   VAR
      sUDT_HMIStatus { ExternalAccessible := 'False'; ExternalVisible := 'False'; ExternalWritable := 'False'; S7_SetPoint := 'False'} : "UDT_WE01Status";   // UDT Weigghing Scale status
      sUDT_Status { ExternalAccessible := 'False'; ExternalVisible := 'False'; ExternalWritable := 'False'; S7_SetPoint := 'False'} : "UDT_CommonStatus";   //  Common status structure
      sUDT_CommonStatus { ExternalAccessible := 'False'; ExternalVisible := 'False'; ExternalWritable := 'False'; S7_SetPoint := 'False'} : "UDT_CommonStatus";   //  Common status structure
      sUDT_CommonStatusOld { ExternalAccessible := 'False'; ExternalVisible := 'False'; ExternalWritable := 'False'; S7_SetPoint := 'False'} : "UDT_CommonStatus";   //  Auxiliary status structure
      sFB_TimerOnOffDelayAutoOn { ExternalAccessible := 'False'; ExternalVisible := 'False'; ExternalWritable := 'False'; S7_SetPoint := 'False'} : "FB_TimerOnOffDelay";
      sx_AutoOnDelayed { ExternalAccessible := 'False'; ExternalVisible := 'False'; ExternalWritable := 'False'} : Bool;
   END_VAR

   VAR CONSTANT
      cdi_DelayOffAutomaticOn : UDInt := 600000;   // Delay before turning off the AutoOn signal
   END_VAR


BEGIN
	(*
	----------------------------------------------------------------------------------------

	Version history:
	Date        | Version   | Author        | Remark
	----------------------------------------------------------------------------------------
	17/09/2019  | 2.0       | M.Singh       | first release TIA 15.1
	21/02/2023  | 4.0       | F.Baten       | 4.0 Release TIA 17.5
	12/03/2024  | 4.1       | S. Nieswie    | Variable name changes accroding to current standard

	 *)

	REGION 1 - Reset Error
	    // If reset Provided from outside; reset the Error

	    IF #iqUDT_EquipmentControl.Command.Reset THEN
	        #sUDT_HMIStatus.Specific.WeighingScaleFault := FALSE;
	    END_IF;
	END_REGION

	REGION 2 - Fault monitoring
	    // Make Camera Error Status

	    IF #ix_ScaleInFault THEN
	        #sUDT_HMIStatus.Specific.WeighingScaleFault := True;
	    END_IF;
	END_REGION

	REGION 3 - Send Automatic Signal to Weighing Scale
	    //  Delay the Turning off of "Automatic on" Signal to Weighing Scale
	    #sFB_TimerOnOffDelayAutoOn(iudi_OffDelayTime := #cdi_DelayOffAutomaticOn,
	                               ix_SignalToDelay := #iqUDT_EquipmentControl.Command.AutomaticOn,
	                               qx_DelayedSignal => #sx_AutoOnDelayed);

	    #qx_Automatic := #sx_AutoOnDelayed;
	END_REGION

	REGION 10 - Make Status
	    // Set Common Status Report

	    // Error active
	    #sUDT_CommonStatus.Error := #sUDT_HMIStatus.Specific.WeighingScaleFault;

	    // Running
	    #sUDT_CommonStatus.Running := #iqUDT_EquipmentControl.Command.AutomaticOn AND NOT #sUDT_CommonStatus.Error;

	    // Stopped
	    #sUDT_CommonStatus.Stopped := NOT #qx_Automatic;

	    IF #sUDT_CommonStatusOld <> #sUDT_CommonStatus                   // update on change
	    THEN

	        // HMI status initialization
	        #sUDT_HMIStatus.Status := 0;

	        // Running in Automatic mode
	        IF #sUDT_CommonStatus.Running
	        THEN
	            #sUDT_HMIStatus.Status := "DB_HMIStatusConfiguration".Running;
	        END_IF;

	        // Stopped
	        IF #sUDT_CommonStatus.Stopped THEN
	            #sUDT_HMIStatus.Status := "DB_HMIStatusConfiguration".Stopped;
	        END_IF;

	        // Error
	        IF #sUDT_HMIStatus.Specific.WeighingScaleFault
	        THEN
	            #sUDT_HMIStatus.Status := "DB_HMIStatusConfiguration".Error;
	        END_IF;

	        #sUDT_CommonStatusOld := #sUDT_CommonStatus;                  // Copy status to memory
	        #sUDT_Status := #sUDT_CommonStatus;                           // Copy status to output
	    END_IF;

	    #qUDT_HMIStatus := #sUDT_HMIStatus;                               // Copy HMI status to output
	    #qUDT_Status := #sUDT_Status;                                     // Copy common status to output


	END_REGION

	REGION 11 - Report to control block

	    // Function to manage report between control block and conveyor block

	    "FC_EquipmentReport"(iUDT_Status := #sUDT_CommonStatus,
	                         iqUDT_Control := #iqUDT_EquipmentControl);

	END_REGION


END_FUNCTION_BLOCK

FUNCTION_BLOCK "FB_MCOConveyLinxAixFullZPA"
TITLE = ConveyLinx reduced ZPA segment
{ S7_Optimized_Access := 'TRUE' }
AUTHOR : 'Ihab Ajram'
FAMILY : ConveyLinx
NAME : ConveyLinx_Reduced_ZPA
VERSION : 0.6
//Version
//history:
//Date        | Version   | Author        | Remark
//----------------------------------------------------------------------------------------
//28/03/2024  | 0.1       | I.Ajram       | Initial
//17/04/2024  | 0.2       | S. Nieswiec   | Changed first scan bit to be taken from DB_Memory;
//                                        | If no initial direction, then set In Forward (region 0.0.2.3)
//
//11/05/2024  | 0.3       | S. Nieswiec   | Changed first scan bit to be taken from DB_Memory;
//                                        | For ConveyStart a transition from 0 to 2 is needed (region 0.3) i did it with your procedure structur check it please
//                                        | To controle whole segment only the GlobalDirAccModeUpstr variable in the first module of the segment is needed
//                                        | If i'm not mistaken direction is set at autoconfiguration and can't be changed by commands. The commands for changing direction
//                                        | only swap the manual mode direction so writing a 5 runs the whole section in reverse and 6 in forward
//
//16/05/2024  | 0.4       | I.Ajram       | Region 0.3 add a check on #qUDT_AixOutputsModuleUpstream.ConveyStopControl/ #qUDT_AixOutputsModuleDownstream.ConveyStopControl
//                                        | if not #cw_ConeyStopDisable, then set it to #cw_ConeyStopDisable and reset to #cw_NormalFunction after 100ms
//
   VAR_INPUT
      iUDT_AixInputsModuleUpstream { ExternalAccessible := 'False'; ExternalVisible := 'False'; ExternalWritable := 'False'} : "UDT_AixZpaFullIN";   // Input structure of conveylinx in ZPA full for the upstream
      iUDT_AixInputsModuleDownstream { ExternalAccessible := 'False'; ExternalVisible := 'False'; ExternalWritable := 'False'} : "UDT_AixZpaFullIN";   // Input structure of conveylinx in ZPA full for the downstream
      ix_SafetyOk { ExternalAccessible := 'False'; ExternalVisible := 'False'; ExternalWritable := 'False'} : Bool;   // TRUE when safety is ok
      ix_24vOk { ExternalAccessible := 'False'; ExternalVisible := 'False'; ExternalWritable := 'False'} : Bool;   // TRUE when 24VDC is healthy
      ix_ReverseDirection { ExternalAccessible := 'False'; ExternalVisible := 'False'; ExternalWritable := 'False'} : Bool;   // FALSE when to run in forward direction and True to run in Reverse direction
   END_VAR

   VAR_OUTPUT
      qUDT_AixOutputsModuleUpstream { ExternalAccessible := 'False'; ExternalVisible := 'False'; ExternalWritable := 'False'} : "UDT_AixZpaFullOUT";   // Output structure of conveylinx in ZPA full for the upstream
      qUDT_AixOutputsModuleDownstream { ExternalAccessible := 'False'; ExternalVisible := 'False'; ExternalWritable := 'False'} : "UDT_AixZpaFullOUT";   // Output structure of conveylinx in ZPA full for the upstream
      qUDT_HMIStatus { ExternalAccessible := 'False'; ExternalVisible := 'False'; ExternalWritable := 'False'} : "UDT_ConveyorStatus";   // HMI status structure
      qUDT_CommonStatus { ExternalAccessible := 'False'; ExternalVisible := 'False'; ExternalWritable := 'False'} : "UDT_CommonStatus";   // Common status structure
   END_VAR

   VAR_IN_OUT
      iqUDT_EquipmentControl : "UDT_EquipmentControl";   // Equipment control structure
      iqUDT_ConveyorCommand : "UDT_ConveyorCommand";   // Conveyor command stucture
      iqUDT_ConveyorInterface : "UDT_ConveyorInterface";   //           Interface structure
      iqUDT_ZPAinterface : "UDT_ZPAinterface";   // Handshake structure in forward direction
      iqUDT_HandShakeUp : "UDT_ConveyorHandshake";   // Upstream handshake structure in forward direction
   END_VAR

   VAR
      sFB_TimerOnOffDelay_GeneralJam { ExternalAccessible := 'False'; ExternalVisible := 'False'; ExternalWritable := 'False'; S7_SetPoint := 'False'} : "FB_TimerOnOffDelay";
      sR_Trig_ix_ReverseDirection {InstructionName := 'R_TRIG'; LibVersion := '1.0'; ExternalAccessible := 'False'; ExternalVisible := 'False'; ExternalWritable := 'False'; S7_SetPoint := 'False'} : R_TRIG;
      sF_Trig_ix_ReverseDirection {InstructionName := 'F_TRIG'; LibVersion := '1.0'; ExternalAccessible := 'False'; ExternalVisible := 'False'; ExternalWritable := 'False'; S7_SetPoint := 'False'} : F_TRIG;
      sR_Trig_ConvCMD_Reverse {InstructionName := 'R_TRIG'; LibVersion := '1.0'; ExternalAccessible := 'False'; ExternalVisible := 'False'; ExternalWritable := 'False'; S7_SetPoint := 'False'} : R_TRIG;
      sF_Trig_ConvCMD_Reverse {InstructionName := 'F_TRIG'; LibVersion := '1.0'; ExternalAccessible := 'False'; ExternalVisible := 'False'; ExternalWritable := 'False'; S7_SetPoint := 'False'} : F_TRIG;
      sR_Trig_ix_PECUpstreamEoS {InstructionName := 'R_TRIG'; LibVersion := '1.0'; ExternalAccessible := 'False'; ExternalVisible := 'False'; ExternalWritable := 'False'; S7_SetPoint := 'False'} : R_TRIG;
      sF_Trig_ix_PECUpstreamEoS {InstructionName := 'F_TRIG'; LibVersion := '1.0'; ExternalAccessible := 'False'; ExternalVisible := 'False'; ExternalWritable := 'False'; S7_SetPoint := 'False'} : F_TRIG;
      sR_Trig_ix_PECUpstreamBoS {InstructionName := 'R_TRIG'; LibVersion := '1.0'; ExternalAccessible := 'False'; ExternalVisible := 'False'; ExternalWritable := 'False'; S7_SetPoint := 'False'} : R_TRIG;
      sF_Trig_ix_PECUpstreamBoS {InstructionName := 'F_TRIG'; LibVersion := '1.0'; ExternalAccessible := 'False'; ExternalVisible := 'False'; ExternalWritable := 'False'; S7_SetPoint := 'False'} : F_TRIG;
      sR_Trig_ix_PECDownStreamEoS {InstructionName := 'R_TRIG'; LibVersion := '1.0'; ExternalAccessible := 'False'; ExternalVisible := 'False'; ExternalWritable := 'False'; S7_SetPoint := 'False'} : R_TRIG;
      sF_Trig_ix_PECDownStreamEoS {InstructionName := 'F_TRIG'; LibVersion := '1.0'; ExternalAccessible := 'False'; ExternalVisible := 'False'; ExternalWritable := 'False'; S7_SetPoint := 'False'} : F_TRIG;
      sR_Trig_ix_PECDownStreamBoS {InstructionName := 'R_TRIG'; LibVersion := '1.0'; ExternalAccessible := 'False'; ExternalVisible := 'False'; ExternalWritable := 'False'; S7_SetPoint := 'False'} : R_TRIG;
      sF_Trig_ix_PECDownStreamBoS {InstructionName := 'F_TRIG'; LibVersion := '1.0'; ExternalAccessible := 'False'; ExternalVisible := 'False'; ExternalWritable := 'False'; S7_SetPoint := 'False'} : F_TRIG;
      sR_TRIG_UpstreamHandshakeRTS {InstructionName := 'R_TRIG'; LibVersion := '1.0'; ExternalAccessible := 'False'; ExternalVisible := 'False'; ExternalWritable := 'False'; S7_SetPoint := 'False'} : R_TRIG;
      sF_TRIG_DownstreamPlcPEC {InstructionName := 'F_TRIG'; LibVersion := '1.0'; ExternalAccessible := 'False'; ExternalVisible := 'False'; ExternalWritable := 'False'; S7_SetPoint := 'False'} : F_TRIG;
      sF_TRIG_UpstreamHandshakeTIP {InstructionName := 'F_TRIG'; LibVersion := '1.0'; ExternalAccessible := 'False'; ExternalVisible := 'False'; ExternalWritable := 'False'; S7_SetPoint := 'False'} : F_TRIG;
      si_previousDownStreamCount { ExternalAccessible := 'False'; ExternalVisible := 'False'; ExternalWritable := 'False'} : Int;
      sx_DownstreamZoneOccupied { ExternalAccessible := 'False'; ExternalVisible := 'False'; ExternalWritable := 'False'} : Bool;
      sx_DownstreamZoneOccupied1 { ExternalAccessible := 'False'; ExternalVisible := 'False'; ExternalWritable := 'False'} : Bool;
   END_VAR
   VAR RETAIN
      sa_Status { ExternalAccessible := 'False'; ExternalVisible := 'False'; ExternalWritable := 'False'} : Struct   // To SCADA and Logic
         UpStream_Module { ExternalAccessible := 'False'; ExternalVisible := 'False'; ExternalWritable := 'False'} : Struct   // Loading Side Local Status
            UpstreamZone { ExternalAccessible := 'False'; ExternalVisible := 'False'; ExternalWritable := 'False'} : Struct
               PEC { ExternalAccessible := 'False'; ExternalVisible := 'False'; ExternalWritable := 'False'} : Bool;
               MotorRunning { ExternalAccessible := 'False'; ExternalVisible := 'False'; ExternalWritable := 'False'} : Bool;
               Busy { ExternalAccessible := 'False'; ExternalVisible := 'False'; ExternalWritable := 'False'} : Bool;
               JamDetected { ExternalAccessible := 'False'; ExternalVisible := 'False'; ExternalWritable := 'False'} : Bool;
            END_STRUCT;
            DownstreamZone { ExternalAccessible := 'False'; ExternalVisible := 'False'; ExternalWritable := 'False'} : Struct
               PEC { ExternalAccessible := 'False'; ExternalVisible := 'False'; ExternalWritable := 'False'} : Bool;
               MotorRunning { ExternalAccessible := 'False'; ExternalVisible := 'False'; ExternalWritable := 'False'} : Bool;
               Busy { ExternalAccessible := 'False'; ExternalVisible := 'False'; ExternalWritable := 'False'} : Bool;
               JamDetected { ExternalAccessible := 'False'; ExternalVisible := 'False'; ExternalWritable := 'False'} : Bool;
            END_STRUCT;
            ArrivalCount { ExternalAccessible := 'False'; ExternalVisible := 'False'; ExternalWritable := 'False'; S7_SetPoint := 'True'} : Int;
            DepartureCount { ExternalAccessible := 'False'; ExternalVisible := 'False'; ExternalWritable := 'False'} : Int;
         END_STRUCT;
         DownStream_Module { ExternalAccessible := 'False'; ExternalVisible := 'False'; ExternalWritable := 'False'} : Struct   // Loading Side Local Status
            UpstreamZone { ExternalAccessible := 'False'; ExternalVisible := 'False'; ExternalWritable := 'False'} : Struct
               PEC { ExternalAccessible := 'False'; ExternalVisible := 'False'; ExternalWritable := 'False'} : Bool;
               MotorRunning { ExternalAccessible := 'False'; ExternalVisible := 'False'; ExternalWritable := 'False'} : Bool;
               Busy { ExternalAccessible := 'False'; ExternalVisible := 'False'; ExternalWritable := 'False'} : Bool;
               JamDetected { ExternalAccessible := 'False'; ExternalVisible := 'False'; ExternalWritable := 'False'} : Bool;
            END_STRUCT;
            DownstreamZone { ExternalAccessible := 'False'; ExternalVisible := 'False'; ExternalWritable := 'False'} : Struct
               PEC { ExternalAccessible := 'False'; ExternalVisible := 'False'; ExternalWritable := 'False'} : Bool;
               MotorRunning { ExternalAccessible := 'False'; ExternalVisible := 'False'; ExternalWritable := 'False'} : Bool;
               Busy { ExternalAccessible := 'False'; ExternalVisible := 'False'; ExternalWritable := 'False'} : Bool;
               JamDetected { ExternalAccessible := 'False'; ExternalVisible := 'False'; ExternalWritable := 'False'} : Bool;
            END_STRUCT;
            ArrivalCount { ExternalAccessible := 'False'; ExternalVisible := 'False'; ExternalWritable := 'False'; S7_SetPoint := 'True'} : Int;
            DepartureCount { ExternalAccessible := 'False'; ExternalVisible := 'False'; ExternalWritable := 'False'} : Int;
         END_STRUCT;
         ZPA_Section { ExternalAccessible := 'False'; ExternalVisible := 'False'; ExternalWritable := 'False'} : Struct
            InForward { ExternalAccessible := 'False'; ExternalVisible := 'False'; ExternalWritable := 'False'} : Bool;
            InReverse { ExternalAccessible := 'False'; ExternalVisible := 'False'; ExternalWritable := 'False'} : Bool;
            NumberOfBoxes { ExternalAccessible := 'False'; ExternalVisible := 'False'; ExternalWritable := 'False'} : Int;
         END_STRUCT;
      END_STRUCT;
   END_VAR
   VAR
      sa_Procedure { ExternalAccessible := 'False'; ExternalVisible := 'False'; ExternalWritable := 'False'} : Struct   // From block interface
         Start { ExternalAccessible := 'False'; ExternalVisible := 'False'; ExternalWritable := 'False'; S7_SetPoint := 'False'} : "UDT_Interface_Signal";
         Stop { ExternalAccessible := 'False'; ExternalVisible := 'False'; ExternalWritable := 'False'} : "UDT_Interface_Signal";
         ReverseDirection { ExternalAccessible := 'False'; ExternalVisible := 'False'; ExternalWritable := 'False'; S7_SetPoint := 'False'} : "UDT_Interface_Signal";
         ForwardDirection { ExternalAccessible := 'False'; ExternalVisible := 'False'; ExternalWritable := 'False'; S7_SetPoint := 'False'} : "UDT_Interface_Signal";
         Reset { ExternalAccessible := 'False'; ExternalVisible := 'False'; ExternalWritable := 'False'} : "UDT_Interface_Signal";
         ClearJamUpstream { ExternalAccessible := 'False'; ExternalVisible := 'False'; ExternalWritable := 'False'} : "UDT_Interface_Signal";
         ClearJamDownstream { ExternalAccessible := 'False'; ExternalVisible := 'False'; ExternalWritable := 'False'} : "UDT_Interface_Signal";
      END_STRUCT;
   END_VAR
   VAR RETAIN
      FLT { ExternalAccessible := 'False'; ExternalVisible := 'False'; ExternalWritable := 'False'} : Struct
         FaultsPresent { ExternalAccessible := 'False'; ExternalVisible := 'False'; ExternalWritable := 'False'} : Bool;
         UpStream_Module { ExternalAccessible := 'False'; ExternalVisible := 'False'; ExternalWritable := 'False'} : Struct
            Module { ExternalAccessible := 'False'; ExternalVisible := 'False'; ExternalWritable := 'False'} : Struct
               ModuleResetFlag { ExternalAccessible := 'False'; ExternalVisible := 'False'; ExternalWritable := 'False'} : Bool;
               ConnectionsNotOK { ExternalAccessible := 'False'; ExternalVisible := 'False'; ExternalWritable := 'False'} : Bool;
            END_STRUCT;
            LeftMotor { ExternalAccessible := 'False'; ExternalVisible := 'False'; ExternalWritable := 'False'} : Struct
               Overheat { ExternalAccessible := 'False'; ExternalVisible := 'False'; ExternalWritable := 'False'} : Bool;
               MaxTorque { ExternalAccessible := 'False'; ExternalVisible := 'False'; ExternalWritable := 'False'} : Bool;
               Short { ExternalAccessible := 'False'; ExternalVisible := 'False'; ExternalWritable := 'False'} : Bool;
               NotConn { ExternalAccessible := 'False'; ExternalVisible := 'False'; ExternalWritable := 'False'} : Bool;
               Overload { ExternalAccessible := 'False'; ExternalVisible := 'False'; ExternalWritable := 'False'} : Bool;
               Stalled { ExternalAccessible := 'False'; ExternalVisible := 'False'; ExternalWritable := 'False'} : Bool;
               BadHall { ExternalAccessible := 'False'; ExternalVisible := 'False'; ExternalWritable := 'False'} : Bool;
               AnyErr { ExternalAccessible := 'False'; ExternalVisible := 'False'; ExternalWritable := 'False'} : Bool;
               OverVoltage { ExternalAccessible := 'False'; ExternalVisible := 'False'; ExternalWritable := 'False'} : Bool;
               LowVoltage { ExternalAccessible := 'False'; ExternalVisible := 'False'; ExternalWritable := 'False'} : Bool;
            END_STRUCT;
            RightMotor { ExternalAccessible := 'False'; ExternalVisible := 'False'; ExternalWritable := 'False'} : Struct
               Overheat { ExternalAccessible := 'False'; ExternalVisible := 'False'; ExternalWritable := 'False'} : Bool;
               MaxTorque { ExternalAccessible := 'False'; ExternalVisible := 'False'; ExternalWritable := 'False'} : Bool;
               Short { ExternalAccessible := 'False'; ExternalVisible := 'False'; ExternalWritable := 'False'} : Bool;
               NotConn { ExternalAccessible := 'False'; ExternalVisible := 'False'; ExternalWritable := 'False'} : Bool;
               Overload { ExternalAccessible := 'False'; ExternalVisible := 'False'; ExternalWritable := 'False'} : Bool;
               Stalled { ExternalAccessible := 'False'; ExternalVisible := 'False'; ExternalWritable := 'False'} : Bool;
               BadHall { ExternalAccessible := 'False'; ExternalVisible := 'False'; ExternalWritable := 'False'} : Bool;
               NotUsed { ExternalAccessible := 'False'; ExternalVisible := 'False'; ExternalWritable := 'False'} : Bool;
               AnyErr { ExternalAccessible := 'False'; ExternalVisible := 'False'; ExternalWritable := 'False'} : Bool;
               OverVoltage { ExternalAccessible := 'False'; ExternalVisible := 'False'; ExternalWritable := 'False'} : Bool;
               LowVoltage { ExternalAccessible := 'False'; ExternalVisible := 'False'; ExternalWritable := 'False'} : Bool;
            END_STRUCT;
            LeftSensor { ExternalAccessible := 'False'; ExternalVisible := 'False'; ExternalWritable := 'False'} : Struct
               LowGain { ExternalAccessible := 'False'; ExternalVisible := 'False'; ExternalWritable := 'False'} : Bool;
               Jam { ExternalAccessible := 'False'; ExternalVisible := 'False'; ExternalWritable := 'False'} : Bool;
            END_STRUCT;
            RightSensor { ExternalAccessible := 'False'; ExternalVisible := 'False'; ExternalWritable := 'False'} : Struct
               LowGain { ExternalAccessible := 'False'; ExternalVisible := 'False'; ExternalWritable := 'False'} : Bool;
               Jam { ExternalAccessible := 'False'; ExternalVisible := 'False'; ExternalWritable := 'False'} : Bool;
            END_STRUCT;
         END_STRUCT;
         DownStream_Module { ExternalAccessible := 'False'; ExternalVisible := 'False'; ExternalWritable := 'False'} : Struct
            Module { ExternalAccessible := 'False'; ExternalVisible := 'False'; ExternalWritable := 'False'} : Struct
               ModuleResetFlag { ExternalAccessible := 'False'; ExternalVisible := 'False'; ExternalWritable := 'False'} : Bool;
               ConnectionsNotOK { ExternalAccessible := 'False'; ExternalVisible := 'False'; ExternalWritable := 'False'} : Bool;
            END_STRUCT;
            LeftMotor { ExternalAccessible := 'False'; ExternalVisible := 'False'; ExternalWritable := 'False'} : Struct
               Overheat { ExternalAccessible := 'False'; ExternalVisible := 'False'; ExternalWritable := 'False'} : Bool;
               MaxTorque { ExternalAccessible := 'False'; ExternalVisible := 'False'; ExternalWritable := 'False'} : Bool;
               Short { ExternalAccessible := 'False'; ExternalVisible := 'False'; ExternalWritable := 'False'} : Bool;
               NotConn { ExternalAccessible := 'False'; ExternalVisible := 'False'; ExternalWritable := 'False'} : Bool;
               Overload { ExternalAccessible := 'False'; ExternalVisible := 'False'; ExternalWritable := 'False'} : Bool;
               Stalled { ExternalAccessible := 'False'; ExternalVisible := 'False'; ExternalWritable := 'False'} : Bool;
               BadHall { ExternalAccessible := 'False'; ExternalVisible := 'False'; ExternalWritable := 'False'} : Bool;
               NotUsed { ExternalAccessible := 'False'; ExternalVisible := 'False'; ExternalWritable := 'False'} : Bool;
               AnyErr { ExternalAccessible := 'False'; ExternalVisible := 'False'; ExternalWritable := 'False'} : Bool;
               OverVoltage { ExternalAccessible := 'False'; ExternalVisible := 'False'; ExternalWritable := 'False'} : Bool;
               LowVoltage { ExternalAccessible := 'False'; ExternalVisible := 'False'; ExternalWritable := 'False'} : Bool;
            END_STRUCT;
            RightMotor { ExternalAccessible := 'False'; ExternalVisible := 'False'; ExternalWritable := 'False'} : Struct
               Overheat { ExternalAccessible := 'False'; ExternalVisible := 'False'; ExternalWritable := 'False'} : Bool;
               MaxTorque { ExternalAccessible := 'False'; ExternalVisible := 'False'; ExternalWritable := 'False'} : Bool;
               Short { ExternalAccessible := 'False'; ExternalVisible := 'False'; ExternalWritable := 'False'} : Bool;
               NotConn { ExternalAccessible := 'False'; ExternalVisible := 'False'; ExternalWritable := 'False'} : Bool;
               Overload { ExternalAccessible := 'False'; ExternalVisible := 'False'; ExternalWritable := 'False'} : Bool;
               Stalled { ExternalAccessible := 'False'; ExternalVisible := 'False'; ExternalWritable := 'False'} : Bool;
               BadHall { ExternalAccessible := 'False'; ExternalVisible := 'False'; ExternalWritable := 'False'} : Bool;
               NotUsed { ExternalAccessible := 'False'; ExternalVisible := 'False'; ExternalWritable := 'False'} : Bool;
               AnyErr { ExternalAccessible := 'False'; ExternalVisible := 'False'; ExternalWritable := 'False'} : Bool;
               OverVoltage { ExternalAccessible := 'False'; ExternalVisible := 'False'; ExternalWritable := 'False'} : Bool;
               LowVoltage { ExternalAccessible := 'False'; ExternalVisible := 'False'; ExternalWritable := 'False'} : Bool;
            END_STRUCT;
            LeftSensor { ExternalAccessible := 'False'; ExternalVisible := 'False'; ExternalWritable := 'False'} : Struct
               LowGain { ExternalAccessible := 'False'; ExternalVisible := 'False'; ExternalWritable := 'False'} : Bool;
               Jam { ExternalAccessible := 'False'; ExternalVisible := 'False'; ExternalWritable := 'False'} : Bool;
            END_STRUCT;
            RightSensor { ExternalAccessible := 'False'; ExternalVisible := 'False'; ExternalWritable := 'False'} : Struct
               LowGain { ExternalAccessible := 'False'; ExternalVisible := 'False'; ExternalWritable := 'False'} : Bool;
               Jam { ExternalAccessible := 'False'; ExternalVisible := 'False'; ExternalWritable := 'False'} : Bool;
            END_STRUCT;
         END_STRUCT;
         GeneralFaults { ExternalAccessible := 'False'; ExternalVisible := 'False'; ExternalWritable := 'False'} : Struct
            GeneralMotorError { ExternalAccessible := 'False'; ExternalVisible := 'False'; ExternalWritable := 'False'} : Bool;   // Stopping motor error somewhere in segment (stalled and max torque not included).
            GeneralNetworkError { ExternalAccessible := 'False'; ExternalVisible := 'False'; ExternalWritable := 'False'} : Bool;   // Network error somewhere in segment
            GeneralJamError { ExternalAccessible := 'False'; ExternalVisible := 'False'; ExternalWritable := 'False'} : Bool;   // JAM error somewhere in segment
            GeneralSensorError { ExternalAccessible := 'False'; ExternalVisible := 'False'; ExternalWritable := 'False'} : Bool;   // Missing sensor somewhere in segment
         END_STRUCT;
      END_STRUCT;
   END_VAR
   VAR
      UpstreamClearJamWDT { ExternalAccessible := 'False'; ExternalVisible := 'False'; ExternalWritable := 'False'; S7_SetPoint := 'False'} : "FB_TimerOnOffDelay";
      DownstreamClearJamWDT { ExternalAccessible := 'False'; ExternalVisible := 'False'; ExternalWritable := 'False'; S7_SetPoint := 'False'} : "FB_TimerOnOffDelay";
      ResetConveyStopControlPulse { ExternalAccessible := 'False'; ExternalVisible := 'False'; ExternalWritable := 'False'; S7_SetPoint := 'False'} : "FB_TimerOnOffDelay";
      si_GinBuffer { ExternalAccessible := 'False'; ExternalVisible := 'False'; ExternalWritable := 'False'} : Int;
      sx_ResetConveyStopControls { ExternalAccessible := 'False'; ExternalVisible := 'False'; ExternalWritable := 'False'} : Bool;
      sx_GinWrote { ExternalAccessible := 'False'; ExternalVisible := 'False'; ExternalWritable := 'False'} : Bool;
      sFB_TimerOnOffDelay_ConveyStopTo0 { ExternalAccessible := 'False'; ExternalVisible := 'False'; ExternalWritable := 'False'; S7_SetPoint := 'False'} : "FB_TimerOnOffDelay";
      sTOF_DownstreamZoneOccupied {InstructionName := 'TOF_TIME'; LibVersion := '1.0'; ExternalAccessible := 'False'; ExternalVisible := 'False'; ExternalWritable := 'False'; S7_SetPoint := 'False'} : TOF_TIME;
   END_VAR

   VAR CONSTANT
      cw_NormalFunction : Word := 0;
      cw_AccumulateZones : Word := 1;
      cw_ChangeAccumulationReleaseMode : Word := 3;
      cw_ReturnReleaseModeToConfiguredDefault : Word := 4;
      cw_RunAllFWDDirection : Word := 5;
      cw_RunAllREVDirection : Word := 6;
      cw_PlaceAllInMaintenanceMode : Word := 7;
      cw_SetDirectionToConfiguredDefaultForward : Word := 10;
      cw_SetDirectionToOppositeOfConfiguredDefaultReverse : Word := 11;
      cw_SelectAllModulesMask : Word := 16#00FF;
      cw_ZoneToWakeUpToAccept : Word := 4;
      cw_ZoneToStopWakeUp : Word := 1;
      cw_ConveyRun : Word := 2;
      cw_ConveyStop : Word := 1;
      cw_ConveyStopDisable : Word := 16#0000;
      cw_ClearJam : Word := 1;   // reset to 0 after jam cleared
      cw_AllowRelease : Word := 1;
      cw_LaneFull : Word := 5;
   END_VAR


BEGIN
	(*
	----------------------------------------------------------------------------------------

	Version
	history:
	Date        | Version   | Author        | Remark
	----------------------------------------------------------------------------------------
	28/03/2024  | 0.1       | I.Ajram       | Initial
	17/04/2024  | 0.2       | S. Nieswiec   | Changed first scan bit to be taken from DB_Memory;
	                                        | If no initial direction, then set In Forward (region 0.0.2.3)

	11/05/2024  | 0.3       | S. Nieswiec   | Changed first scan bit to be taken from DB_Memory;
	                                        | For ConveyStart a transition from 0 to 2 is needed (region 0.3) i did it with your procedure structur check it please
	                                        | To controle whole segment only the GlobalDirAccModeUpstr variable in the first module of the segment is needed
	                                        | If i'm not mistaken direction is set at autoconfiguration and can't be changed by commands. The commands for changing direction
	                                        | only swap the manual mode direction so writing a 5 runs the whole section in reverse and 6 in forward

	16/05/2024  | 0.4       | I.Ajram       | Region 0.3 add a check on #qUDT_AixOutputsModuleUpstream.ConveyStopControl/ #qUDT_AixOutputsModuleDownstream.ConveyStopControl
	                                        | if not #cw_ConeyStopDisable, then set it to #cw_ConeyStopDisable and reset to #cw_NormalFunction after 100ms
	                                        | activated IEC check on FB
	22/05/2024  | 0.5       | S. Nieswiec   | Added PECs from plc conveyors upstream and downstream to block interface
	                                        | Rewrote handshake logic (region 5)
	                                        | Added general errors (region 3.3)

	05/06/2024  | 0.6       | S. Nieswiec   | Changes regarding conveystop
	02/10/2024  | 0.7       | R. Willems    | Moved downstream signals to new function block in downstream zone sequence, and handle signals between both blocks
	                                          Added PEC interface handling upstream zone and downstream zone



	*)
	REGION 0 Block interface
	    REGION 0.0.1 edge detection
	        #sR_Trig_ix_ReverseDirection(CLK := #ix_ReverseDirection);
	        #sR_Trig_ConvCMD_Reverse(CLK := #iqUDT_ConveyorCommand.Reverse);
	        #sF_Trig_ix_ReverseDirection(CLK := #ix_ReverseDirection);
	        #sF_Trig_ConvCMD_Reverse(CLK := #iqUDT_ConveyorCommand.Reverse);
	        #sR_Trig_ix_PECUpstreamEoS(CLK := #iUDT_AixInputsModuleUpstream.AllSensorPortInputs.RightSensor);
	        #sF_Trig_ix_PECUpstreamEoS(CLK := #iUDT_AixInputsModuleUpstream.AllSensorPortInputs.RightSensor);
	        #sR_Trig_ix_PECUpstreamBoS(CLK := #iUDT_AixInputsModuleUpstream.AllSensorPortInputs.LeftSensor);
	        #sF_Trig_ix_PECUpstreamBoS(CLK := #iUDT_AixInputsModuleUpstream.AllSensorPortInputs.LeftSensor);
	        #sR_Trig_ix_PECDownStreamEoS(CLK := #iUDT_AixInputsModuleDownstream.AllSensorPortInputs.RightSensor);
	        #sF_Trig_ix_PECDownStreamEoS(CLK := #iUDT_AixInputsModuleDownstream.AllSensorPortInputs.RightSensor);
	        #sR_Trig_ix_PECDownStreamBoS(CLK := #iUDT_AixInputsModuleDownstream.AllSensorPortInputs.LeftSensor);
	        #sF_Trig_ix_PECDownStreamBoS(CLK := #iUDT_AixInputsModuleDownstream.AllSensorPortInputs.LeftSensor);
	        #sR_TRIG_UpstreamHandshakeRTS(CLK := #iqUDT_HandShakeUp.RTS);
	        IF (#iUDT_AixInputsModuleDownstream.DepartureCountDownstreamZone <> #iUDT_AixInputsModuleDownstream.ArrivalCountDownstreamZone) THEN
	            #sx_DownstreamZoneOccupied1 := TRUE;
	        ELSE
	            #sx_DownstreamZoneOccupied1 := FALSE;
	        END_IF;
	        #sTOF_DownstreamZoneOccupied(IN := #sx_DownstreamZoneOccupied1,
	                                     PT := T#500ms,
	                                     Q => #sx_DownstreamZoneOccupied);

	        #sF_TRIG_DownstreamPlcPEC(CLK := #sx_DownstreamZoneOccupied);
	        #sF_TRIG_UpstreamHandshakeTIP(CLK := #iqUDT_HandShakeUp.TIP);



	    END_REGION
	    REGION 0.0.2 Initial Conditions
	        REGION 0.0.2.1 in Forward
	            IF #sa_Status.ZPA_Section.InForward THEN
	                IF "DB_Memory".FirstScan THEN
	                    #qUDT_AixOutputsModuleDownstream.SetDishargeStatus := #cw_LaneFull;
	                    // ToDo add additional initial conditions here
	                END_IF;
	            END_IF;
	        END_REGION
	        REGION 0.0.2.2 in Reverse
	            IF #sa_Status.ZPA_Section.InReverse THEN
	                IF "DB_Memory".FirstScan THEN
	                    #qUDT_AixOutputsModuleUpstream.SetDishargeStatus := #cw_LaneFull;
	                    // ToDo add additional initial conditions here
	                END_IF;
	            END_IF;
	        END_REGION
	        REGION 0.0.2.3 no initial direction - set into Forward
	            IF NOT #sa_Status.ZPA_Section.InReverse AND NOT #sa_Status.ZPA_Section.InForward THEN

	                #sa_Status.ZPA_Section.InForward := TRUE;

	            END_IF;

	        END_REGION

	    END_REGION
	    REGION 0.1 Forward
	        REGION 0.1.2  Request
	            IF (NOT #sa_Status.ZPA_Section.InForward AND
	                (#sF_Trig_ix_ReverseDirection.Q OR #sF_Trig_ConvCMD_Reverse.Q)
	                ) OR
	                ("DB_Memory".FirstScan AND #sa_Status.ZPA_Section.InForward)
	            THEN
	                #sa_Procedure.ForwardDirection.RQST := TRUE;
	            END_IF;
	        END_REGION
	        REGION 0.1.3 Command
	            IF #sa_Procedure.ForwardDirection.RQST AND
	                #iqUDT_EquipmentControl.Report.Stopped
	            THEN
	                #sa_Procedure.ForwardDirection.CMD := TRUE;
	                #sa_Procedure.ForwardDirection.RQST := FALSE;
	            END_IF;
	        END_REGION
	        REGION 0.1.4 Set direction Forward
	            IF #sa_Procedure.ForwardDirection.CMD THEN
	                #qUDT_AixOutputsModuleUpstream.GlobalDirAccModeUpstr :=
	                #cw_SetDirectionToConfiguredDefaultForward AND 16#00FF;
	                #sa_Procedure.ForwardDirection.CMD := FALSE;
	                #sa_Status.ZPA_Section.InForward := TRUE;
	                #sa_Status.ZPA_Section.InReverse := FALSE;
	            END_IF;
	        END_REGION
	    END_REGION
	    REGION 0.2 Reverse

	        REGION 0.2.2  Request
	            IF (NOT #sa_Status.ZPA_Section.InReverse AND
	                (#sR_Trig_ix_ReverseDirection.Q OR #sR_Trig_ConvCMD_Reverse.Q)
	                ) OR
	                ("DB_Memory".FirstScan AND #sa_Status.ZPA_Section.InReverse)
	            THEN
	                #sa_Procedure.ReverseDirection.RQST := TRUE;
	            END_IF;
	        END_REGION
	        REGION 0.2.3 Command
	            IF #sa_Procedure.ReverseDirection.RQST AND
	                #iqUDT_EquipmentControl.Report.Stopped
	            THEN
	                #sa_Procedure.ReverseDirection.CMD := TRUE;
	                #sa_Procedure.ReverseDirection.RQST := FALSE;
	            END_IF;
	        END_REGION
	        REGION 0.2.4 set direction Reverse
	            IF #sa_Procedure.ReverseDirection.CMD THEN
	                #qUDT_AixOutputsModuleUpstream.GlobalDirAccModeUpstr :=
	                #cw_SetDirectionToOppositeOfConfiguredDefaultReverse AND 16#00FF;
	                #sa_Procedure.ReverseDirection.CMD := FALSE;
	                #sa_Status.ZPA_Section.InForward := FALSE;
	                #sa_Status.ZPA_Section.InReverse := TRUE;
	            END_IF;
	        END_REGION
	    END_REGION
	    REGION 0.3 Start

	        IF #iqUDT_EquipmentControl.Command.Start THEN
	            #sa_Procedure.Start.RQST := TRUE;
	        END_IF;

	        IF #sa_Procedure.Start.RQST THEN
	            IF #qUDT_AixOutputsModuleUpstream.ConveyStopControl <> #cw_ConveyStopDisable OR
	                #qUDT_AixOutputsModuleDownstream.ConveyStopControl <> #cw_ConveyStopDisable
	            THEN
	                #qUDT_AixOutputsModuleUpstream.ConveyStopControl := #cw_ConveyStopDisable;
	                #qUDT_AixOutputsModuleDownstream.ConveyStopControl := #cw_ConveyStopDisable;
	                #sx_ResetConveyStopControls := TRUE;
	            END_IF;
	            IF #ResetConveyStopControlPulse.qx_DelayedSignal OR
	                NOT #sx_ResetConveyStopControls
	            THEN
	                #sx_ResetConveyStopControls := FALSE;
	                #sa_Procedure.Start.CMD := TRUE;
	                #sa_Procedure.Start.RQST := FALSE;
	            END_IF;
	        END_IF;

	        #ResetConveyStopControlPulse(ix_Enable := TRUE,
	                                     ix_SignalToDelay := #sx_ResetConveyStopControls,
	                                     iudi_OffDelayTime := 0,
	                                     iudi_OnDelayTime := 100);


	        IF #sa_Procedure.Start.CMD THEN
	            #qUDT_AixOutputsModuleUpstream.GlobalDirAccModeUpstr := #cw_NormalFunction;

	            #qUDT_AixOutputsModuleUpstream.ConveyStopControl := #cw_ConveyRun;
	            #qUDT_AixOutputsModuleDownstream.ConveyStopControl := #cw_ConveyRun;
	            #sa_Procedure.Start.CMD := FALSE;
	        END_IF;
	    END_REGION
	    REGION 0.4 Stop
	        REGION 0.4.1 Stop request
	            IF (#iqUDT_EquipmentControl.Command.Stop
	                OR #sa_Procedure.ForwardDirection.RQST
	                OR #sa_Procedure.ReverseDirection.RQST
	                OR #FLT.FaultsPresent)
	                AND NOT (#qUDT_AixOutputsModuleUpstream.ConveyStopControl = #cw_ConveyStop)

	            THEN
	                #sa_Procedure.Stop.RQST := TRUE;
	            END_IF;
	        END_REGION
	        REGION 0.4.2 Stop command
	            IF #sa_Procedure.Stop.RQST
	                AND NOT #iqUDT_HandShakeUp.TIP
	                AND NOT #iqUDT_ZPAinterface.Handshake.TIP
	            THEN
	                #qUDT_AixOutputsModuleUpstream.ConveyStopControl := #cw_ConveyStop;
	                #qUDT_AixOutputsModuleDownstream.ConveyStopControl := #cw_ConveyStop;
	                #sa_Procedure.Stop.RQST := FALSE;
	            END_IF;
	        END_REGION

	        #sFB_TimerOnOffDelay_ConveyStopTo0(iudi_OnDelayTime := 1000,
	                                           ix_SignalToDelay := #qUDT_AixOutputsModuleDownstream.ConveyStopControl = #cw_ConveyStop,
	                                           ix_Enable := TRUE);

	        IF #sFB_TimerOnOffDelay_ConveyStopTo0.qx_DelayedSignal THEN
	            #qUDT_AixOutputsModuleDownstream.ConveyStopControl := 0;
	            #qUDT_AixOutputsModuleUpstream.ConveyStopControl := 0;
	        END_IF;

	    END_REGION
	END_REGION

	REGION 1 Reset faults

	    REGION 1.1 - Send reset request to interface UDT

	        // Reset signal is sent to the interface UDT (VFD block, Tracking block, PEC update block)
	        #iqUDT_ConveyorInterface.InternalErrorReset := #iqUDT_EquipmentControl.Command.Reset;
	        #iqUDT_ZPAinterface.ConveyorInterface.InternalErrorReset := #iqUDT_EquipmentControl.Command.Reset;
	        #iqUDT_ConveyorInterface.ResetStatistics := #iqUDT_EquipmentControl.Command.ResetData;
	        #iqUDT_ZPAinterface.ConveyorInterface.ResetStatistics := #iqUDT_EquipmentControl.Command.ResetData;

	    END_REGION

	END_REGION
	REGION 2 Local Status
	    IF #sa_Status.ZPA_Section.InForward THEN
	        REGION 2.2 Status specific for Forward Direction
	            REGION 2.2.1 Up stream Module
	                REGION 2.2.1.1 Up Stream Zone
	                    #sa_Status.UpStream_Module.UpstreamZone.PEC :=
	                    #iUDT_AixInputsModuleUpstream.LocalUpstreamZoneStatus_Fwd = 16#04 OR
	                    #iUDT_AixInputsModuleUpstream.LocalUpstreamZoneStatus_Fwd = 16#05;

	                    #sa_Status.UpStream_Module.UpstreamZone.MotorRunning :=
	                    #iUDT_AixInputsModuleUpstream.LocalUpstreamZoneStatus_Fwd = 16#02 OR
	                    #iUDT_AixInputsModuleUpstream.LocalUpstreamZoneStatus_Fwd = 16#04;

	                    #sa_Status.UpStream_Module.UpstreamZone.Busy :=
	                    #iUDT_AixInputsModuleUpstream.LocalUpstreamZoneStatus_Fwd = 16#06;

	                END_REGION
	                REGION 2.2.1.2 Down Stream Zone
	                    #sa_Status.UpStream_Module.DownstreamZone.PEC :=
	                    #iUDT_AixInputsModuleUpstream.LocalDownstreamZoneStatus_Fwd = 16#04 OR
	                    #iUDT_AixInputsModuleUpstream.LocalDownstreamZoneStatus_Fwd = 16#05;

	                    #sa_Status.UpStream_Module.DownstreamZone.MotorRunning :=
	                    #iUDT_AixInputsModuleUpstream.LocalDownstreamZoneStatus_Fwd = 16#02 OR
	                    #iUDT_AixInputsModuleUpstream.LocalDownstreamZoneStatus_Fwd = 16#04;

	                    #sa_Status.UpStream_Module.DownstreamZone.Busy :=
	                    #iUDT_AixInputsModuleUpstream.LocalDownstreamZoneStatus_Fwd = 16#06;
	                END_REGION
	                REGION 2.2.1.3 Arrival / Departure count
	                    #sa_Status.UpStream_Module.ArrivalCount := #iUDT_AixInputsModuleUpstream.ArrivalCountUpstreamZone;
	                    #sa_Status.UpStream_Module.DepartureCount := #iUDT_AixInputsModuleUpstream.DepartureCountDownstreamZone;
	                END_REGION
	            END_REGION
	            REGION 2.2.2 Down stream Module
	                REGION 2.2.2.1 Up Stream Zone
	                    #sa_Status.DownStream_Module.UpstreamZone.PEC :=
	                    #iUDT_AixInputsModuleDownstream.LocalUpstreamZoneStatus_Fwd = 16#04 OR
	                    #iUDT_AixInputsModuleDownstream.LocalUpstreamZoneStatus_Fwd = 16#05;

	                    #sa_Status.DownStream_Module.UpstreamZone.MotorRunning :=
	                    #iUDT_AixInputsModuleDownstream.LocalUpstreamZoneStatus_Fwd = 16#02 OR
	                    #iUDT_AixInputsModuleDownstream.LocalUpstreamZoneStatus_Fwd = 16#04;

	                    #sa_Status.DownStream_Module.UpstreamZone.Busy :=
	                    #iUDT_AixInputsModuleDownstream.LocalUpstreamZoneStatus_Fwd = 16#06;
	                END_REGION
	                REGION 2.2.2.2 Down Stream Zone
	                    #sa_Status.DownStream_Module.DownstreamZone.PEC :=
	                    #iUDT_AixInputsModuleDownstream.LocalDownstreamZoneStatus_Fwd = 16#04 OR
	                    #iUDT_AixInputsModuleDownstream.LocalDownstreamZoneStatus_Fwd = 16#05;

	                    #sa_Status.DownStream_Module.DownstreamZone.MotorRunning :=
	                    #iUDT_AixInputsModuleDownstream.LocalDownstreamZoneStatus_Fwd = 16#02 OR
	                    #iUDT_AixInputsModuleDownstream.LocalDownstreamZoneStatus_Fwd = 16#04;

	                    #sa_Status.DownStream_Module.DownstreamZone.Busy :=
	                    #iUDT_AixInputsModuleDownstream.LocalDownstreamZoneStatus_Fwd = 16#06;
	                END_REGION
	                REGION 2.2.2.3 Arrival / Departure count
	                    #sa_Status.DownStream_Module.ArrivalCount := #iUDT_AixInputsModuleDownstream.ArrivalCountUpstreamZone;
	                    #sa_Status.DownStream_Module.DepartureCount := #iUDT_AixInputsModuleDownstream.DepartureCountDownstreamZone;
	                END_REGION
	            END_REGION
	            REGION 2.2.3 ZPA section Box Count
	                #sa_Status.ZPA_Section.NumberOfBoxes := #sa_Status.UpStream_Module.ArrivalCount - #sa_Status.DownStream_Module.DepartureCount;
	            END_REGION
	        END_REGION
	    ELSIF #sa_Status.ZPA_Section.InReverse THEN
	        REGION 2.3 Status specific for Reverse Direction
	            REGION 2.3.1 Up stream Module
	                REGION 2.3.1.1 Up Stream Zone
	                    #sa_Status.UpStream_Module.UpstreamZone.PEC :=
	                    #iUDT_AixInputsModuleUpstream.LocalUpstreamZoneStatus_Rev = 16#04 OR
	                    #iUDT_AixInputsModuleUpstream.LocalUpstreamZoneStatus_Rev = 16#05;

	                    #sa_Status.UpStream_Module.UpstreamZone.MotorRunning :=
	                    #iUDT_AixInputsModuleUpstream.LocalUpstreamZoneStatus_Rev = 16#02 OR
	                    #iUDT_AixInputsModuleUpstream.LocalUpstreamZoneStatus_Rev = 16#04;

	                    #sa_Status.UpStream_Module.UpstreamZone.Busy :=
	                    #iUDT_AixInputsModuleUpstream.LocalUpstreamZoneStatus_Rev = 16#06;
	                END_REGION
	                REGION 2.3.1.2 Down Stream Zone
	                    #sa_Status.UpStream_Module.DownstreamZone.PEC :=
	                    #iUDT_AixInputsModuleUpstream.LocalDownstreamZoneStatus_Rev = 16#04 OR
	                    #iUDT_AixInputsModuleUpstream.LocalDownstreamZoneStatus_Rev = 16#05;

	                    #sa_Status.UpStream_Module.DownstreamZone.MotorRunning :=
	                    #iUDT_AixInputsModuleUpstream.LocalDownstreamZoneStatus_Rev = 16#02 OR
	                    #iUDT_AixInputsModuleUpstream.LocalDownstreamZoneStatus_Rev = 16#04;

	                    #sa_Status.UpStream_Module.DownstreamZone.Busy :=
	                    #iUDT_AixInputsModuleUpstream.LocalDownstreamZoneStatus_Rev = 16#06;
	                END_REGION
	                REGION 2.3.1.3 Arrival / Departure count
	                    #sa_Status.UpStream_Module.ArrivalCount := #iUDT_AixInputsModuleUpstream.ArrivalCountDownstreamZone;
	                    #sa_Status.UpStream_Module.DepartureCount := #iUDT_AixInputsModuleUpstream.DepartureCountUpstreamZone;
	                END_REGION
	            END_REGION
	            REGION 2.3.2 Down stream Module
	                REGION 2.3.2.1 Up Stream Zone
	                    #sa_Status.DownStream_Module.UpstreamZone.PEC :=
	                    #iUDT_AixInputsModuleDownstream.LocalUpstreamZoneStatus_Rev = 16#04 OR
	                    #iUDT_AixInputsModuleDownstream.LocalUpstreamZoneStatus_Rev = 16#05;

	                    #sa_Status.DownStream_Module.UpstreamZone.MotorRunning :=
	                    #iUDT_AixInputsModuleDownstream.LocalUpstreamZoneStatus_Rev = 16#02 OR
	                    #iUDT_AixInputsModuleDownstream.LocalUpstreamZoneStatus_Rev = 16#04;

	                    #sa_Status.DownStream_Module.UpstreamZone.Busy :=
	                    #iUDT_AixInputsModuleDownstream.LocalUpstreamZoneStatus_Rev = 16#06;
	                END_REGION
	                REGION 2.3.2.2 Down Stream Zone
	                    #sa_Status.DownStream_Module.DownstreamZone.PEC :=
	                    #iUDT_AixInputsModuleDownstream.LocalDownstreamZoneStatus_Rev = 16#04 OR
	                    #iUDT_AixInputsModuleDownstream.LocalDownstreamZoneStatus_Rev = 16#05;

	                    #sa_Status.DownStream_Module.DownstreamZone.MotorRunning :=
	                    #iUDT_AixInputsModuleDownstream.LocalDownstreamZoneStatus_Rev = 16#02 OR
	                    #iUDT_AixInputsModuleDownstream.LocalDownstreamZoneStatus_Rev = 16#04;

	                    #sa_Status.DownStream_Module.DownstreamZone.Busy :=
	                    #iUDT_AixInputsModuleDownstream.LocalDownstreamZoneStatus_Rev = 16#06;
	                END_REGION
	                REGION 2.3.2.3 Arrival / Departure count
	                    #sa_Status.DownStream_Module.ArrivalCount := #iUDT_AixInputsModuleDownstream.ArrivalCountDownstreamZone;
	                    #sa_Status.DownStream_Module.DepartureCount := #iUDT_AixInputsModuleDownstream.DepartureCountUpstreamZone;
	                END_REGION
	            END_REGION
	            REGION 2.3.3 ZPA section Box Count
	                #sa_Status.ZPA_Section.NumberOfBoxes := #sa_Status.DownStream_Module.ArrivalCount - #sa_Status.UpStream_Module.DepartureCount;
	            END_REGION

	        END_REGION
	    END_IF;
	    REGION 2.4 Equipment Report
	        REGION 2.4.1 Stopped
	            #iqUDT_EquipmentControl.Report.Stopped :=
	            #iUDT_AixInputsModuleUpstream.ConveyStopStatus.StopActiveCommandPLC OR
	            #iUDT_AixInputsModuleUpstream.ConveyStopStatus.StopActiveOtherModule OR
	            #iUDT_AixInputsModuleDownstream.ConveyStopStatus.StopActiveCommandPLC OR
	            #iUDT_AixInputsModuleDownstream.ConveyStopStatus.StopActiveOtherModule OR
	            FALSE;
	        END_REGION
	        REGION 2.4.1 Halted
	            #iqUDT_EquipmentControl.Report.Halted :=
	            #iUDT_AixInputsModuleUpstream.ConveyStopStatus.StopActiveLostConn OR
	            #iUDT_AixInputsModuleUpstream.ConveyStopStatus.StopActiveLostPLC OR
	            #iUDT_AixInputsModuleDownstream.ConveyStopStatus.StopActiveLostConn OR
	            #iUDT_AixInputsModuleDownstream.ConveyStopStatus.StopActiveLostPLC OR
	            FALSE;
	        END_REGION
	        REGION 2.4.2 Safety Stop
	            #iqUDT_EquipmentControl.Report.SafetyStop :=
	            NOT #ix_SafetyOk;
	        END_REGION
	        REGION 2.4.3 Warning
	            #iqUDT_EquipmentControl.Report.Warning :=
	            #FLT.UpStream_Module.LeftSensor.LowGain OR
	            #FLT.UpStream_Module.RightSensor.LowGain OR
	            #FLT.DownStream_Module.LeftSensor.LowGain OR
	            #FLT.DownStream_Module.RightSensor.LowGain;
	        END_REGION
	        REGION 2.4.4 Manual
	            #iqUDT_EquipmentControl.Report.Manual :=
	            (
	            #qUDT_AixOutputsModuleUpstream.GlobalDirAccModeDnstr = #cw_RunAllFWDDirection OR
	            #qUDT_AixOutputsModuleUpstream.GlobalDirAccModeDnstr = #cw_RunAllREVDirection
	            ) OR
	            (
	            #qUDT_AixOutputsModuleUpstream.GlobalDirAccModeUpstr = #cw_RunAllFWDDirection OR
	            #qUDT_AixOutputsModuleUpstream.GlobalDirAccModeUpstr = #cw_RunAllREVDirection
	            ) OR
	            (
	            #qUDT_AixOutputsModuleDownstream.GlobalDirAccModeDnstr = #cw_RunAllFWDDirection OR
	            #qUDT_AixOutputsModuleDownstream.GlobalDirAccModeDnstr = #cw_RunAllREVDirection
	            ) OR
	            (
	            #qUDT_AixOutputsModuleDownstream.GlobalDirAccModeUpstr = #cw_RunAllFWDDirection OR
	            #qUDT_AixOutputsModuleDownstream.GlobalDirAccModeUpstr = #cw_RunAllREVDirection
	            ) OR
	            FALSE;
	        END_REGION
	        REGION 2.4.5 Running
	            #iqUDT_EquipmentControl.Report.Running := NOT #iqUDT_EquipmentControl.Report.Stopped;
	        END_REGION
	        REGION 2.4.6 Manual Running
	            #iqUDT_EquipmentControl.Report.ManualRun :=
	            #iqUDT_EquipmentControl.Report.Running AND
	            #iqUDT_EquipmentControl.Report.Manual;
	        END_REGION
	        REGION 2.4.7 Energy Save
	            // ZPA is always in energy save
	            #iqUDT_EquipmentControl.Report.EnergySave := TRUE;
	        END_REGION
	        REGION 2.4.8 AutoON
	            #iqUDT_EquipmentControl.Report.AutoON := #iqUDT_EquipmentControl.Report.Running;
	        END_REGION
	        REGION 2.4.9 Error
	            #iqUDT_EquipmentControl.Report.Error :=
	            #FLT.FaultsPresent OR
	            FALSE;
	        END_REGION
	        REGION 2.4.10 Jam detection
	            #sa_Status.UpStream_Module.UpstreamZone.JamDetected := #iUDT_AixInputsModuleUpstream.Diagnostic.UpstreamJamErr;
	            #sa_Status.UpStream_Module.DownstreamZone.JamDetected := #iUDT_AixInputsModuleUpstream.Diagnostic.DownstreamJamErr;
	            #sa_Status.DownStream_Module.UpstreamZone.JamDetected := #iUDT_AixInputsModuleDownstream.Diagnostic.UpstreamJamErr;
	            #sa_Status.DownStream_Module.DownstreamZone.JamDetected := #iUDT_AixInputsModuleDownstream.Diagnostic.DownstreamJamErr;


	        END_REGION
	        REGION 2.4.11 Pass Reset Signal to Module
	            REGION 2.4.11.1 Reset Request
	                IF #iqUDT_EquipmentControl.Command.Reset AND
	                    #iqUDT_EquipmentControl.Report.Error
	                THEN
	                    #sa_Procedure.Reset.RQST := TRUE;
	                END_IF;
	            END_REGION
	            REGION 2.4.11.2 Reset Command
	                IF #sa_Procedure.Reset.RQST AND
	                    NOT #iqUDT_EquipmentControl.Report.Running
	                THEN
	                    #sa_Procedure.Reset.RQST := FALSE;

	                    // upstream
	                    #qUDT_AixOutputsModuleUpstream.ClearMotorError := 1;
	                    #qUDT_AixOutputsModuleUpstream.ClearJamUpstream := 1;
	                    #qUDT_AixOutputsModuleUpstream.ClearJamDownstream := 1;
	                    // downstream
	                    #qUDT_AixOutputsModuleDownstream.ClearMotorError := 1;
	                    #qUDT_AixOutputsModuleDownstream.ClearJamUpstream := 1;
	                    #qUDT_AixOutputsModuleDownstream.ClearJamDownstream := 1;
	                END_IF;
	            END_REGION
	        END_REGION
	        REGION 2.4.12 Upstream Pass Clear Jam Signal to Module
	            REGION 2.4.12.1 Upstream Clear Jam Request
	                IF #iqUDT_EquipmentControl.Command.Reset AND
	                    (#sa_Status.UpStream_Module.UpstreamZone.JamDetected OR
	                    #sa_Status.UpStream_Module.DownstreamZone.JamDetected)
	                THEN
	                    #sa_Procedure.ClearJamUpstream.RQST := TRUE;
	                END_IF;
	            END_REGION
	            REGION 2.4.12.2 Upstream ClearJam Command
	                IF #sa_Procedure.ClearJamUpstream.RQST
	                THEN
	                    #sa_Procedure.ClearJamUpstream.RQST := FALSE;
	                    #sa_Procedure.ClearJamUpstream.CMD := TRUE;
	                    #qUDT_AixOutputsModuleUpstream.ClearJamUpstream := 1;
	                    #qUDT_AixOutputsModuleUpstream.ClearJamDownstream := 1;
	                END_IF;
	            END_REGION
	            REGION 2.4.12.3 Upstream ClearJamWDT
	                #UpstreamClearJamWDT(iudi_OnDelayTime := 6000,
	                                     iudi_OffDelayTime := 0,
	                                     ix_Enable := TRUE,
	                                     ix_SignalToDelay := #sa_Procedure.ClearJamUpstream.CMD);
	            END_REGION
	            REGION 2.4.12.4 Upstream Exit Clear Jam
	                IF NOT (#sa_Status.UpStream_Module.UpstreamZone.JamDetected OR
	                    #sa_Status.UpStream_Module.DownstreamZone.JamDetected)
	                    OR #UpstreamClearJamWDT.qx_DelayedSignal
	                THEN
	                    #qUDT_AixOutputsModuleUpstream.ClearJamUpstream := 0;
	                    #qUDT_AixOutputsModuleUpstream.ClearJamDownstream := 0;
	                    #sa_Procedure.ClearJamUpstream.CMD := FALSE;
	                END_IF;
	            END_REGION
	        END_REGION
	        REGION 2.4.13 Downstream Pass Clear Jam Signal to Module
	            REGION 2.4.13.1 downstream Clear Jam Request
	                IF #iqUDT_EquipmentControl.Command.Reset AND
	                    (#sa_Status.DownStream_Module.UpstreamZone.JamDetected OR
	                    #sa_Status.DownStream_Module.DownstreamZone.JamDetected)
	                THEN
	                    #sa_Procedure.ClearJamDownstream.RQST := TRUE;
	                END_IF;
	            END_REGION
	            REGION 2.4.13.2 downstream ClearJam Command
	                IF #sa_Procedure.ClearJamDownstream.RQST
	                THEN
	                    #sa_Procedure.ClearJamDownstream.RQST := FALSE;
	                    #sa_Procedure.ClearJamDownstream.CMD := TRUE;
	                    #qUDT_AixOutputsModuleDownstream.ClearJamUpstream := 1;
	                    #qUDT_AixOutputsModuleDownstream.ClearJamDownstream := 1;
	                END_IF;
	            END_REGION
	            REGION 2.4.13.3 downstream ClearJamWDT
	                #DownstreamClearJamWDT(iudi_OnDelayTime := 6000,
	                                       iudi_OffDelayTime := 0,
	                                       ix_Enable := TRUE,
	                                       ix_SignalToDelay := #sa_Procedure.ClearJamDownstream.CMD);
	            END_REGION
	            REGION 2.4.13.4 downstream Exit Clear Jam
	                IF NOT (#sa_Status.DownStream_Module.UpstreamZone.JamDetected OR
	                    #sa_Status.DownStream_Module.DownstreamZone.JamDetected)
	                    OR #DownstreamClearJamWDT.qx_DelayedSignal
	                THEN
	                    #qUDT_AixOutputsModuleDownstream.ClearJamUpstream := 0;
	                    #qUDT_AixOutputsModuleDownstream.ClearJamDownstream := 0;
	                    #sa_Procedure.ClearJamDownstream.CMD := FALSE;
	                END_IF;
	            END_REGION
	        END_REGION
	    END_REGION
	END_REGION

	REGION 3 Faults
	    REGION 3.0 Faults present detection

	        #FLT.FaultsPresent := #FLT.UpStream_Module.Module.ConnectionsNotOK
	        OR #FLT.UpStream_Module.LeftMotor.AnyErr
	        OR #FLT.UpStream_Module.RightMotor.AnyErr
	        OR #FLT.UpStream_Module.LeftSensor.LowGain
	        OR #FLT.UpStream_Module.RightSensor.LowGain
	        //  OR #FLT.UpStream_Module.LeftSensor.Jam
	        //  OR #FLT.UpStream_Module.RightSensor.Jam

	        OR #FLT.DownStream_Module.Module.ConnectionsNotOK
	        OR #FLT.DownStream_Module.LeftMotor.AnyErr
	        OR #FLT.DownStream_Module.RightMotor.AnyErr
	        OR #FLT.DownStream_Module.LeftSensor.LowGain
	        OR #FLT.DownStream_Module.RightSensor.LowGain
	        // OR #FLT.DownStream_Module.LeftSensor.Jam
	        // OR #FLT.DownStream_Module.RightSensor.Jam

	        OR #FLT.GeneralFaults.GeneralMotorError
	        OR #FLT.GeneralFaults.GeneralNetworkError
	        OR #FLT.GeneralFaults.GeneralJamError
	        OR #FLT.GeneralFaults.GeneralSensorError

	        OR #iqUDT_ConveyorInterface.InternalErrorPEC
	        OR #iqUDT_ZPAinterface.ConveyorInterface.InternalErrorPEC
	        OR FALSE;

	    END_REGION

	    REGION 3.1 UpStream
	        REGION 3.1.1 Module

	            #FLT.UpStream_Module.Module.ModuleResetFlag := #iUDT_AixInputsModuleUpstream.Diagnostic.ModuleResetFlag;

	            IF #iUDT_AixInputsModuleUpstream.Diagnostic.ConnectionsNotOK THEN
	                #FLT.UpStream_Module.Module.ConnectionsNotOK := TRUE;
	            END_IF;
	        END_REGION
	        REGION 3.1.2 Left Motor

	            IF #iUDT_AixInputsModuleUpstream.Diagnostic.LeftMotorOverheat THEN
	                #FLT.UpStream_Module.LeftMotor.Overheat := TRUE;
	            END_IF;

	            IF #iUDT_AixInputsModuleUpstream.Diagnostic.LeftMotorMaxTorque THEN
	                #FLT.UpStream_Module.LeftMotor.MaxTorque := TRUE;
	            END_IF;

	            IF #iUDT_AixInputsModuleUpstream.Diagnostic.LeftMotorShort THEN
	                #FLT.UpStream_Module.LeftMotor.Short := TRUE;
	            END_IF;

	            IF #iUDT_AixInputsModuleUpstream.Diagnostic.LeftMotorNotConn THEN
	                #FLT.UpStream_Module.LeftMotor.NotConn := TRUE;
	            END_IF;

	            IF #iUDT_AixInputsModuleUpstream.Diagnostic.LeftMotorOverload THEN
	                #FLT.UpStream_Module.LeftMotor.Overload := TRUE;
	            END_IF;

	            IF #iUDT_AixInputsModuleUpstream.Diagnostic.LeftMotorStalled THEN
	                #FLT.UpStream_Module.LeftMotor.Stalled := TRUE;
	            END_IF;

	            IF #iUDT_AixInputsModuleUpstream.Diagnostic.LeftMotorBadHall THEN
	                #FLT.UpStream_Module.LeftMotor.BadHall := TRUE;
	            END_IF;

	            IF #iUDT_AixInputsModuleUpstream.Diagnostic.LeftMotorAnyErr THEN
	                #FLT.UpStream_Module.LeftMotor.AnyErr := TRUE;
	            END_IF;

	            IF #iUDT_AixInputsModuleUpstream.Diagnostic.OverVoltage THEN
	                #FLT.UpStream_Module.LeftMotor.OverVoltage := TRUE;
	            END_IF;

	            IF #iUDT_AixInputsModuleUpstream.Diagnostic.LowVoltage THEN
	                #FLT.UpStream_Module.LeftMotor.LowVoltage := TRUE;
	            END_IF;
	        END_REGION

	        REGION 3.1.3 Right Motor

	            IF #iUDT_AixInputsModuleUpstream.Diagnostic.RightMotorOverheat THEN
	                #FLT.UpStream_Module.RightMotor.Overheat := TRUE;
	            END_IF;

	            IF #iUDT_AixInputsModuleUpstream.Diagnostic.RightMotorMaxTorque THEN
	                #FLT.UpStream_Module.RightMotor.MaxTorque := TRUE;
	            END_IF;

	            IF #iUDT_AixInputsModuleUpstream.Diagnostic.RightMotorShort THEN
	                #FLT.UpStream_Module.RightMotor.Short := TRUE;
	            END_IF;

	            IF #iUDT_AixInputsModuleUpstream.Diagnostic.RightMotorNotConn THEN
	                #FLT.UpStream_Module.RightMotor.NotConn := TRUE;
	            END_IF;

	            IF #iUDT_AixInputsModuleUpstream.Diagnostic.RightMotorOverload THEN
	                #FLT.UpStream_Module.RightMotor.Overload := TRUE;
	            END_IF;

	            IF #iUDT_AixInputsModuleUpstream.Diagnostic.RightMotorStalled THEN
	                #FLT.UpStream_Module.RightMotor.Stalled := TRUE;
	            END_IF;

	            IF #iUDT_AixInputsModuleUpstream.Diagnostic.RightMotorBadHall THEN
	                #FLT.UpStream_Module.RightMotor.BadHall := TRUE;
	            END_IF;

	            IF #iUDT_AixInputsModuleUpstream.Diagnostic.RightMotorAnyErr THEN
	                #FLT.UpStream_Module.RightMotor.AnyErr := TRUE;
	            END_IF;

	            IF #iUDT_AixInputsModuleUpstream.Diagnostic.OverVoltage THEN
	                #FLT.UpStream_Module.RightMotor.OverVoltage := TRUE;
	            END_IF;

	            IF #iUDT_AixInputsModuleUpstream.Diagnostic.LowVoltage THEN
	                #FLT.UpStream_Module.RightMotor.LowVoltage := TRUE;
	            END_IF;

	        END_REGION
	        REGION 3.1.4 Left Sensor
	            IF #iUDT_AixInputsModuleUpstream.Diagnostic.LeftSensLowGain THEN
	                #FLT.UpStream_Module.LeftSensor.LowGain := TRUE;
	            END_IF;

	            IF #sa_Status.UpStream_Module.UpstreamZone.JamDetected
	                AND NOT #sa_Procedure.ClearJamUpstream.CMD
	                AND NOT #sa_Procedure.ClearJamUpstream.RQST
	            THEN
	                #FLT.UpStream_Module.LeftSensor.Jam := TRUE;
	            ELSE
	                #FLT.UpStream_Module.LeftSensor.Jam := FALSE;
	            END_IF;
	        END_REGION
	        REGION 3.1.5 Right Sensor
	            IF #iUDT_AixInputsModuleUpstream.Diagnostic.RightSensLowGain THEN
	                #FLT.UpStream_Module.RightSensor.LowGain := TRUE;
	            END_IF;

	            IF #sa_Status.UpStream_Module.DownstreamZone.JamDetected
	                AND NOT #sa_Procedure.ClearJamUpstream.CMD
	                AND NOT #sa_Procedure.ClearJamUpstream.RQST
	            THEN
	                #FLT.UpStream_Module.RightSensor.Jam := TRUE;
	            ELSE
	                #FLT.UpStream_Module.RightSensor.Jam := FALSE;
	            END_IF;
	        END_REGION
	    END_REGION

	    REGION 3.2 DownStream
	        REGION 3.2.1 Module

	            #FLT.DownStream_Module.Module.ModuleResetFlag := #iUDT_AixInputsModuleDownstream.Diagnostic.ModuleResetFlag;

	            IF #iUDT_AixInputsModuleDownstream.Diagnostic.ConnectionsNotOK THEN
	                #FLT.DownStream_Module.Module.ConnectionsNotOK := TRUE;
	            END_IF;
	        END_REGION
	        REGION 3.2.2 Left Motor

	            IF #iUDT_AixInputsModuleDownstream.Diagnostic.LeftMotorOverheat THEN
	                #FLT.DownStream_Module.LeftMotor.Overheat := TRUE;
	            END_IF;

	            IF #iUDT_AixInputsModuleDownstream.Diagnostic.LeftMotorMaxTorque THEN
	                #FLT.DownStream_Module.LeftMotor.MaxTorque := TRUE;
	            END_IF;

	            IF #iUDT_AixInputsModuleDownstream.Diagnostic.LeftMotorShort THEN
	                #FLT.DownStream_Module.LeftMotor.Short := TRUE;
	            END_IF;

	            IF #iUDT_AixInputsModuleDownstream.Diagnostic.LeftMotorNotConn THEN
	                #FLT.DownStream_Module.LeftMotor.NotConn := TRUE;
	            END_IF;

	            IF #iUDT_AixInputsModuleDownstream.Diagnostic.LeftMotorOverload THEN
	                #FLT.DownStream_Module.LeftMotor.Overload := TRUE;
	            END_IF;

	            IF #iUDT_AixInputsModuleDownstream.Diagnostic.LeftMotorStalled THEN
	                #FLT.DownStream_Module.LeftMotor.Stalled := TRUE;
	            END_IF;

	            IF #iUDT_AixInputsModuleDownstream.Diagnostic.LeftMotorBadHall THEN
	                #FLT.DownStream_Module.LeftMotor.BadHall := TRUE;
	            END_IF;

	            IF #iUDT_AixInputsModuleDownstream.Diagnostic.LeftMotorAnyErr THEN
	                #FLT.DownStream_Module.LeftMotor.AnyErr := TRUE;
	            END_IF;

	            IF #iUDT_AixInputsModuleDownstream.Diagnostic.OverVoltage THEN
	                #FLT.DownStream_Module.LeftMotor.OverVoltage := TRUE;
	            END_IF;

	            IF #iUDT_AixInputsModuleDownstream.Diagnostic.LowVoltage THEN
	                #FLT.DownStream_Module.LeftMotor.LowVoltage := TRUE;
	            END_IF;
	        END_REGION

	        REGION 3.2.3 Right Motor

	            IF #iUDT_AixInputsModuleDownstream.Diagnostic.RightMotorOverheat THEN
	                #FLT.DownStream_Module.RightMotor.Overheat := TRUE;
	            END_IF;

	            IF #iUDT_AixInputsModuleDownstream.Diagnostic.RightMotorMaxTorque THEN
	                #FLT.DownStream_Module.RightMotor.MaxTorque := TRUE;
	            END_IF;

	            IF #iUDT_AixInputsModuleDownstream.Diagnostic.RightMotorShort THEN
	                #FLT.DownStream_Module.RightMotor.Short := TRUE;
	            END_IF;

	            IF #iUDT_AixInputsModuleDownstream.Diagnostic.RightMotorNotConn THEN
	                #FLT.DownStream_Module.RightMotor.NotConn := TRUE;
	            END_IF;

	            IF #iUDT_AixInputsModuleDownstream.Diagnostic.RightMotorOverload THEN
	                #FLT.DownStream_Module.RightMotor.Overload := TRUE;
	            END_IF;

	            IF #iUDT_AixInputsModuleDownstream.Diagnostic.RightMotorStalled THEN
	                #FLT.DownStream_Module.RightMotor.Stalled := TRUE;
	            END_IF;

	            IF #iUDT_AixInputsModuleDownstream.Diagnostic.RightMotorBadHall THEN
	                #FLT.DownStream_Module.RightMotor.BadHall := TRUE;
	            END_IF;

	            IF #iUDT_AixInputsModuleDownstream.Diagnostic.RightMotorAnyErr THEN
	                #FLT.DownStream_Module.RightMotor.AnyErr := TRUE;
	            END_IF;

	            IF #iUDT_AixInputsModuleDownstream.Diagnostic.OverVoltage THEN
	                #FLT.DownStream_Module.RightMotor.OverVoltage := TRUE;
	            END_IF;

	            IF #iUDT_AixInputsModuleDownstream.Diagnostic.LowVoltage THEN
	                #FLT.DownStream_Module.RightMotor.LowVoltage := TRUE;
	            END_IF;

	        END_REGION
	        REGION 3.2.4 Left Sensor
	            IF #iUDT_AixInputsModuleDownstream.Diagnostic.LeftSensLowGain THEN
	                #FLT.DownStream_Module.LeftSensor.LowGain := TRUE;
	            END_IF;

	            IF #sa_Status.DownStream_Module.UpstreamZone.JamDetected
	                AND NOT #sa_Procedure.ClearJamUpstream.CMD
	                AND NOT #sa_Procedure.ClearJamUpstream.RQST
	            THEN
	                #FLT.DownStream_Module.LeftSensor.Jam := TRUE;
	            ELSE
	                #FLT.DownStream_Module.LeftSensor.Jam := FALSE;
	            END_IF;
	        END_REGION
	        REGION 3.2.5 Right Sensor
	            IF #iUDT_AixInputsModuleDownstream.Diagnostic.RightSensLowGain THEN
	                #FLT.DownStream_Module.RightSensor.LowGain := TRUE;
	            END_IF;

	            IF #sa_Status.DownStream_Module.DownstreamZone.JamDetected
	                AND NOT #sa_Procedure.ClearJamDownstream.CMD
	                AND NOT #sa_Procedure.ClearJamDownstream.RQST
	            THEN
	                #FLT.DownStream_Module.RightSensor.Jam := TRUE;
	            ELSE
	                #FLT.DownStream_Module.RightSensor.Jam := FALSE;
	            END_IF;
	        END_REGION
	    END_REGION

	    REGION 3.3 General
	        // Error present somewhere in whole segment

	        REGION 3.3.1 Motor error
	            IF #iUDT_AixInputsModuleDownstream.GeneralLineError.MotorError THEN
	                #FLT.GeneralFaults.GeneralMotorError := TRUE;
	            END_IF;
	        END_REGION


	        REGION 3.3.2 Network error
	            IF #iUDT_AixInputsModuleDownstream.GeneralLineError.ConnectionError THEN
	                #FLT.GeneralFaults.GeneralNetworkError := TRUE;
	            END_IF;
	        END_REGION

	        REGION 3.3.3 Jam error

	            #sFB_TimerOnOffDelay_GeneralJam(iudi_OnDelayTime := 500,
	                                            ix_SignalToDelay := #iUDT_AixInputsModuleDownstream.GeneralLineError.JamError
	                                            AND #qUDT_AixOutputsModuleUpstream.ConveyStopControl = #cw_ConveyRun,
	                                            ix_Enable := TRUE);

	            IF #sFB_TimerOnOffDelay_GeneralJam.qx_DelayedSignal
	                AND NOT #sa_Procedure.ClearJamDownstream.RQST
	                AND NOT #sa_Procedure.ClearJamUpstream.RQST
	                AND #qUDT_AixOutputsModuleUpstream.ConveyStopControl = #cw_ConveyRun
	            THEN
	                #FLT.GeneralFaults.GeneralJamError := TRUE;

	            ELSIF #iqUDT_EquipmentControl.Command.Reset AND (#qUDT_AixOutputsModuleUpstream.ConveyStopControl = 0) THEN
	                #FLT.GeneralFaults.GeneralJamError := FALSE;
	            END_IF;
	        END_REGION

	        REGION 3.3.4 Sensor Error
	            IF #iUDT_AixInputsModuleDownstream.GeneralLineError.MotorError THEN
	                #FLT.GeneralFaults.GeneralSensorError := TRUE;
	            END_IF;
	        END_REGION

	    END_REGION

	    REGION 3.4 - Error Resets
	        IF #iqUDT_EquipmentControl.Command.Reset THEN

	            #FLT.UpStream_Module.Module.ConnectionsNotOK := FALSE;
	            #FLT.UpStream_Module.LeftMotor.Overheat := FALSE;
	            #FLT.UpStream_Module.LeftMotor.MaxTorque := FALSE;
	            #FLT.UpStream_Module.LeftMotor.Short := FALSE;
	            #FLT.UpStream_Module.LeftMotor.NotConn := FALSE;
	            #FLT.UpStream_Module.LeftMotor.Overload := FALSE;
	            #FLT.UpStream_Module.LeftMotor.Stalled := FALSE;
	            #FLT.UpStream_Module.LeftMotor.BadHall := FALSE;
	            #FLT.UpStream_Module.LeftMotor.AnyErr := FALSE;
	            #FLT.UpStream_Module.LeftMotor.OverVoltage := FALSE;
	            #FLT.UpStream_Module.LeftMotor.LowVoltage := FALSE;
	            #FLT.UpStream_Module.RightMotor.Overheat := FALSE;
	            #FLT.UpStream_Module.RightMotor.MaxTorque := FALSE;
	            #FLT.UpStream_Module.RightMotor.Short := FALSE;
	            #FLT.UpStream_Module.RightMotor.NotConn := FALSE;
	            #FLT.UpStream_Module.RightMotor.Overload := FALSE;
	            #FLT.UpStream_Module.RightMotor.Stalled := FALSE;
	            #FLT.UpStream_Module.RightMotor.BadHall := FALSE;
	            #FLT.UpStream_Module.RightMotor.AnyErr := FALSE;
	            #FLT.UpStream_Module.RightMotor.OverVoltage := FALSE;
	            #FLT.UpStream_Module.RightMotor.LowVoltage := FALSE;
	            #FLT.UpStream_Module.LeftSensor.LowGain := FALSE;
	            #FLT.UpStream_Module.RightSensor.LowGain := FALSE;


	            #FLT.DownStream_Module.Module.ConnectionsNotOK := FALSE;
	            #FLT.DownStream_Module.LeftMotor.Overheat := FALSE;
	            #FLT.DownStream_Module.LeftMotor.MaxTorque := FALSE;
	            #FLT.DownStream_Module.LeftMotor.Short := FALSE;
	            #FLT.DownStream_Module.LeftMotor.NotConn := FALSE;
	            #FLT.DownStream_Module.LeftMotor.Overload := FALSE;
	            #FLT.DownStream_Module.LeftMotor.Stalled := FALSE;
	            #FLT.DownStream_Module.LeftMotor.BadHall := FALSE;
	            #FLT.DownStream_Module.LeftMotor.AnyErr := FALSE;
	            #FLT.DownStream_Module.LeftMotor.OverVoltage := FALSE;
	            #FLT.DownStream_Module.LeftMotor.LowVoltage := FALSE;
	            #FLT.DownStream_Module.RightMotor.Overheat := FALSE;
	            #FLT.DownStream_Module.RightMotor.MaxTorque := FALSE;
	            #FLT.DownStream_Module.RightMotor.Short := FALSE;
	            #FLT.DownStream_Module.RightMotor.NotConn := FALSE;
	            #FLT.DownStream_Module.RightMotor.Overload := FALSE;
	            #FLT.DownStream_Module.RightMotor.Stalled := FALSE;
	            #FLT.DownStream_Module.RightMotor.BadHall := FALSE;
	            #FLT.DownStream_Module.RightMotor.AnyErr := FALSE;
	            #FLT.DownStream_Module.RightMotor.OverVoltage := FALSE;
	            #FLT.DownStream_Module.RightMotor.LowVoltage := FALSE;
	            #FLT.DownStream_Module.LeftSensor.LowGain := FALSE;
	            #FLT.DownStream_Module.RightSensor.LowGain := FALSE;

	            #FLT.GeneralFaults.GeneralMotorError := FALSE;
	            #FLT.GeneralFaults.GeneralSensorError := FALSE;
	            #FLT.GeneralFaults.GeneralNetworkError := FALSE;
	            //  #FLT.GeneralFaults.GeneralJamError := FALSE;

	            #iqUDT_ConveyorInterface.InternalErrorPEC := FALSE;
	            #iqUDT_ZPAinterface.ConveyorInterface.InternalErrorPEC := FALSE;

	        END_IF;

	    END_REGION
	END_REGION


	REGION 4 HandShake
	    IF #iqUDT_EquipmentControl.Report.Running THEN
	        REGION 4.1 Forward direction
	            IF #sa_Status.ZPA_Section.InForward THEN


	                REGION 4.1.2 Request received from upstream conveyor
	                    // if module is sleeping empty and upstream is requesting to send then wake up module
	                    IF #iUDT_AixInputsModuleUpstream.LocalUpstreamZoneStatus_Fwd = 16#01 AND NOT #iqUDT_HandShakeUp.RTS THEN

	                        #qUDT_AixOutputsModuleUpstream.SetInductStatus := #cw_ZoneToWakeUpToAccept;
	                    ELSE
	                        #qUDT_AixOutputsModuleUpstream.SetInductStatus := #cw_ZoneToStopWakeUp;
	                    END_IF;
	                END_REGION ;


	                REGION 4.1.1 RTR ready to receive
	                    // If module is running empty waiting for parcel and no jams are present then send RTR
	                    IF #iUDT_AixInputsModuleUpstream.LocalUpstreamZoneStatus_Fwd = 16#02
	                        AND NOT #sa_Status.UpStream_Module.UpstreamZone.JamDetected
	                        AND NOT #sa_Status.UpStream_Module.DownstreamZone.JamDetected
	                    THEN
	                        #iqUDT_HandShakeUp.RTR := TRUE;
	                    ELSE
	                        #iqUDT_HandShakeUp.RTR := FALSE;
	                    END_IF;
	                END_REGION


	                REGION 4.1.2 Box transfer from PLC to ZPA conveyor

	                    // When parcel left PLC controlled conveyor and there was GIN in handshake the write it into buffer and set flag
	                    IF #sR_TRIG_UpstreamHandshakeRTS.Q AND #iqUDT_HandShakeUp.GIN <> 0 THEN

	                        #qUDT_AixOutputsModuleUpstream.InductTrackingOnUpstreamZone := INT_TO_DWORD(#iqUDT_HandShakeUp.GIN);
	                        #sx_GinWrote := TRUE;
	                    END_IF;

	                    //If there was GIN in handshake and parcel reaches Upstream zone PEC then accept tracking data
	                    IF #sx_GinWrote AND #sR_Trig_ix_PECUpstreamBoS.Q THEN

	                        #qUDT_AixOutputsModuleUpstream.SetReleaseCountUpstream += 1;  // No protection needed, works after overshoot
	                        #sx_GinWrote := FALSE;

	                    END_IF;

	                    // Reset handshake data after TIP ends
	                    IF #sF_TRIG_UpstreamHandshakeTIP.Q THEN
	                        #iqUDT_HandShakeUp.NrOfPosToShift := 0;
	                    END_IF;
	                END_REGION


	                REGION 4.1.4 Send RTS and copy tracking data into buffer when parcel arrives at PEC
	                    IF #sR_Trig_ix_PECDownStreamEoS.Q THEN  // what if jam happens, RTS falls down, but product stays on pec the whole time? needs better condition
	                        #iqUDT_ZPAinterface.Handshake.RTS := TRUE; // is being set to true, but goes to false into the same cycle when rtr present
	                        #si_GinBuffer := DWORD_TO_INT(#iUDT_AixInputsModuleDownstream.TrackingDownstreamZone);
	                    END_IF;
	                END_REGION


	                REGION 4.1.5 Start transfer on RTR and RTS
	                    // Release parcel if RTR is present

	                    IF #iqUDT_ZPAinterface.Handshake.RTR AND #iqUDT_ZPAinterface.Handshake.RTS AND NOT #iqUDT_ZPAinterface.Handshake.TIP AND #sx_DownstreamZoneOccupied THEN

	                        #qUDT_AixOutputsModuleDownstream.SetDishargeStatus := #cw_AllowRelease;
	                        #iqUDT_ZPAinterface.Handshake.TIP := TRUE;
	                        #iqUDT_ZPAinterface.Handshake.RTS := FALSE;

	                    END_IF;
	                END_REGION

	                REGION 4.1.6 Write Gin into handshake when parcel leaves zone
	                    IF #si_GinBuffer <> 0 AND #sF_Trig_ix_PECDownStreamEoS.Q THEN
	                        #iqUDT_ZPAinterface.Handshake.GIN := #si_GinBuffer;
	                        #si_GinBuffer := 0;
	                    END_IF;
	                END_REGION

	                REGION 4.1.7 Box arrives on downstream conveyor and TIP ends
	                    IF #iqUDT_ZPAinterface.Handshake.TIP AND #sF_TRIG_DownstreamPlcPEC.Q
	                    THEN
	                        #iqUDT_ZPAinterface.Handshake.GIN := 0;
	                        #iqUDT_ZPAinterface.Handshake.TIP := FALSE;
	                        #qUDT_AixOutputsModuleDownstream.SetDishargeStatus := #cw_LaneFull;
	                    END_IF;
	                END_REGION

	            END_IF;
	        END_REGION
	    ELSE
	        #iqUDT_HandShakeUp.RTR := FALSE;
	    END_IF;
	END_REGION

	(* //         REGION 4.2 Reverse direction
	//             IF #sa_Status.ZPA_Section.InForward THEN
	//                 REGION 4.2.1 RTR ready to receive
	//                     #iqUDT_HandShake.RTR :=
	//                     #sa_Status.DownStream_Module.DepartureCount = #sa_Status.DownStream_Module.ArrivalCount AND
	//                     NOT (
	//                     #sa_Status.DownStream_Module.UpstreamZone.JamDetected OR
	//                     #sa_Status.DownStream_Module.DownstreamZone.JamDetected
	//                     );
	//                 END_REGION
	//                 REGION 4.2.2 RTS recieved from upstream conveyor
	//                     // if module is RTR and Downstream is requesting to send then wake up module
	//                     IF #iqUDT_HandShake.RTR // AND
	//                        // #iqUDT_HandShakeup.RTS
	//                     THEN
	//                         #qUDT_AixOutputsModuleDownstream.SetInductStatus := #cw_ZoneToRunToAccept;
	//                         #iqUDT_HandShake.TIP := TRUE;
	//                     END_IF;
	//                 END_REGION
	//                 REGION 4.2.3 box Exit Upstream zone

	//                     IF #iqUDT_HandShake.TIP AND
	//                         #sR_Trig_ix_PECDownStreamBoS.Q        // PEC EoS is TRUE if clear
	//                     THEN
	//                         #iqUDT_HandShake.RTR := FALSE;
	//                         #qUDT_AixOutputsModuleDownstream.InductTrackingOnUpstreamZone := INT_TO_DWORD(#iqUDT_HandShakeUp.GIN);
	//                         #qUDT_AixOutputsModuleDownstream.SetInductStatus := #cw_ZoneToAcceptTheTrackingData;
	//                     END_IF;
	//                 END_REGION
	//                 REGION 4.2.4 Send RTS
	//                     IF #sa_Status.UpStream_Module.ArrivalCount > #sa_Status.UpStream_Module.DepartureCount THEN
	//                         #iqUDT_HandShakeUp.RTS := TRUE;
	//                     END_IF;
	//                 END_REGION
	//                 REGION 4.2.5 Start transfer on RTR and RTS

	//                     IF #iqUDT_HandShakeUp.RTR AND #iqUDT_HandShakeUp.RTS
	//                     THEN
	//                         #qUDT_AixOutputsModuleUpstream.SetDishargeStatus := #cw_AllowRelease;
	//                         #iqUDT_HandShakeUp.TIP := TRUE;
	//                         #iqUDT_HandShakeUp.RTS := FALSE;
	//                     END_IF;
	//                 END_REGION
	//                 REGION 4.2.6 Box arrives on downstream conveyor and TIP ends
	//                     IF #iqUDT_HandShakeUp.TIP AND #sF_Trig_ix_PECUpstreamBoS.Q
	//                     THEN
	//                         #iqUDT_HandShakeUp.TIP := FALSE;
	//                         #qUDT_AixOutputsModuleUpstream.SetDishargeStatus := #cw_LaneFull;
	//                     END_IF;
	//                 END_REGION
	//             END_IF;
	//         END_REGION
	//     END_IF; *)  //reverse direction if needed needs to be rewritten

	REGION 5 Actual speed
	    //#si_ActualSpeed := REAL_TO_INT(INT_TO_REAL(WORD_TO_INT(#iUDT_AixInputsModule.RightMotorActualSpeed & #cw_ActualSpeedMask)) * #iUDT_AixConfig.Motor.Ratio);

	END_REGION

	REGION 5 Populate qUDT_Status
	    #qUDT_CommonStatus := #iqUDT_EquipmentControl.Report;
	    #iqUDT_ZPAinterface.CommonStatus := #iqUDT_EquipmentControl.Report;
	END_REGION

END_FUNCTION_BLOCK

FUNCTION "FC_CopyTrackingArray" : Void
{ S7_Optimized_Access := 'TRUE' }
VERSION : 0.1
// ATTRIBUTES
// AUTO_NUMBER = True
// BLOCK_NUMBER = 15
// END_ATTRIBUTES
   VAR_INPUT
      Ix_ConveyorToGlobal : Bool;   // True when data to be moved to global array; FALSE when data to be moved to conveyor array
      ix_FirstConveyor : Bool;   // True when it is first conveyor to global tracking array
      ii_StartPosition : Int;
      ii_Displacement : Int;
      ii_ConveyorLength : DInt;
   END_VAR

   VAR_IN_OUT
      iqs_ConveyorArray : Array[*] of Int;   // Tracking array
      iqs_GlobalArray : Array[*] of Int;   // Tracking array
      iqUDT_EmptyWindow : "UDT_EmptyWindow";
   END_VAR

   VAR_TEMP
      ti_LoopCounter : Int;
      ti_EmptyWindowArrayLength : Int;
   END_VAR


BEGIN
	(*
	----------------------------------------------------------------------------------------
	|                                                                                      |
	|  Copyright  2019             MHS                                                     |
	|  All Rights Rese9ved         Larenweg 90                                             |
	|                              5234 KC 's-Hertogenbosch,                               |
	|                              Netherlands                                             |
	|                                                                                      |
	----------------------------------------------------------------------------------------

	Version history:
	Date        | Version   | Author        | Remark
	----------------------------------------------------------------------------------------
	 29/08/2023 | 3.0       | S. Deulkar    | first release MHS TIA 17
	 13/03/2024 | 4.1       | S. Nieswiec   | first release TIA 18
	*)

	REGION 1 - Copy data from conveyor array to global array

	    IF #Ix_ConveyorToGlobal
	    THEN
	        MOVE_BLK(IN := #iqs_ConveyorArray[0],
	                 COUNT := DINT_TO_ULINT(#ii_ConveyorLength / 10),
	                 OUT => #iqs_GlobalArray[#ii_StartPosition]);
	    END_IF;

	END_REGION

	REGION 2 - Copy data from global array to conveyor array

	    IF NOT #Ix_ConveyorToGlobal
	    THEN
	        MOVE_BLK(IN := #iqs_GlobalArray[#ii_StartPosition],
	                 COUNT := DINT_TO_ULINT(#ii_ConveyorLength / 10),
	                 OUT => #iqs_ConveyorArray[0]);
	    END_IF;

	END_REGION

	REGION 3 - Update empty window position

	    IF #Ix_ConveyorToGlobal
	    THEN
	        #ti_EmptyWindowArrayLength := "FC_GetNrOfArrayEl"(#iqUDT_EmptyWindow.EmptyWIndowPosition);

	        // Update window position with displacement of the conveyor
	        IF (#iqUDT_EmptyWindow.No_Of_Empty_Window > 0)
	            AND (#ii_Displacement > 0)
	        THEN

	            FOR #ti_LoopCounter := 1 TO #iqUDT_EmptyWindow.No_Of_Empty_Window DO

	                IF ((#iqUDT_EmptyWindow.EmptyWIndowPosition[#ti_LoopCounter] >= #ii_StartPosition)
	                    AND (#iqUDT_EmptyWindow.EmptyWIndowPosition[#ti_LoopCounter] <= (#ii_StartPosition + (#ii_ConveyorLength / 10))))

	                THEN
	                    #iqUDT_EmptyWindow.EmptyWIndowPosition[#ti_LoopCounter] -= #ii_Displacement;
	                END_IF;

	            END_FOR;

	        END_IF;

	    END_IF;

	    // IF #ix_FirstConveyor
	    // THEN

	    //     FOR #ti_LoopCounter := #ii_StartPosition TO #ii_StartPosition + #ii_ConveyorLength DO

	    //         IF #iqs_GlobalArray[#ti_LoopCounter] = -100
	    //             AND (#iq_UDT_EmptyWindow.No_Of_Empty_Window + 1) <= #ti_EmptyWindowArrayLength
	    //         THEN
	    //             #iq_UDT_EmptyWindow.No_Of_Empty_Window += 1;
	    //             #iq_UDT_EmptyWindow.EmptyWIndowPosition[#iq_UDT_EmptyWindow.No_Of_Empty_Window + 1] := #ti_LoopCounter;
	    //         END_IF;

	    //     END_FOR;

	    //     // Remove unused empty window from arrat when it pass last induct position
	    //     IF #iq_UDT_EmptyWindow.No_Of_Empty_Window > 0
	    //         AND #iq_UDT_EmptyWindow.EmptyWIndowPosition[1] <= 10
	    //     THEN
	    //         // //Remove used emty window from array
	    //         MOVE_BLK(IN := #iq_UDT_EmptyWindow.EmptyWIndowPosition[2],
	    //                  COUNT := INT_TO_ULINT(#ti_EmptyWindowArrayLength - 1),
	    //                  OUT => #iq_UDT_EmptyWindow.EmptyWIndowPosition[1]);
	    //         #iq_UDT_EmptyWindow.No_Of_Empty_Window -= 1;
	    //     END_IF;

	    // END_IF;

	END_REGION

END_FUNCTION

